Fanuc TP program (LS listing): PRLIFT.LS

/PROG  PRLIFT
/ATTR
OWNER		= MNEDITOR;
COMMENT		= "PrLift";
PROG_SIZE	= 0;
CREATE		= DATE 26-01-01  TIME 00:00:00;
MODIFIED	= DATE 26-01-01  TIME 00:00:00;
FILE_NAME	= ;
VERSION		= 0;
LINE_COUNT	= 5;
MEMORY_SIZE	= 0;
PROTECT		= READ_WRITE;
TCD:  STACK_SIZE	= 0,
      TASK_PRIORITY	= 50,
      TIME_SLICE	= 0,
      BUSY_LAMP_OFF	= 0,
      ABORT_REQUEST	= 0,
      PAUSE_REQUEST	= 0;
DEFAULT_GROUP	= 1,*,*,*,*;
CONTROL_CODE	= 00000000 00000000;
/MN
   1:  !RAPID PointRefProbe.PrLift ;
   2:  PR[98,3]=PR[98,3]-AR[1]    ;
   3:  PR[99]=PR[98]    ;
   4:  CALL PRSHIFT    ;
   5:  PR[98]=PR[99]    ;
/POS
/END
